{attribute 'enable_dynamic_creation'}
{attribute 'no_explicit_call' := 'direct call for this function block is not allowed'}
FUNCTION_BLOCK FB_ErrorTimestamp IMPLEMENTS I_ErrorTimestamp
VAR
	_nTimestamp : ULINT;
END_VAR

// Retrieves the timestamp as a combined date and time value.
METHOD AsDateTime : DT // The combined date and time value as a DT (Date and Time).
VAR_INPUT
END_VAR
AsDateTime := TO_DT(THIS^._nTimestamp/1000);
END_METHOD

// Retrieves the date part of the timestamp.
METHOD GetDate : DATE // The date part of the timestamp.
VAR_INPUT
END_VAR
GetDate := TO_DATE(THIS^._nTimestamp/1000);
END_METHOD

// Retrieves the time of day part of the timestamp.
METHOD GetTimeOfDay : TOD // The time of day part of the timestamp.
VAR_INPUT
END_VAR
GetTimeOfDay := TO_TOD(THIS^._nTimestamp MOD 86400000);
END_METHOD

// The raw timestamp value which represents the number of milliseconds since Thursday, 1.1.1970 00:00:00.000.
// [get] Returns the raw timestamp value.
// [set] Sets the raw timestamp value.
PROPERTY Raw : ULINT
GET
Raw := THIS^._nTimestamp;
END_GET
SET
THIS^._nTimestamp := Raw;
END_SET
END_PROPERTY

END_FUNCTION_BLOCK

(* stored: Version 1.1.0.1
   POU FB_ErrorTimestamp: Id {3006405e-b4c3-05aa-13ca-bc7db81a079f}, SpecialFunc None
   Method AsDateTime: Id {f8abec48-c1cf-0a93-07f7-ae776de09770}
   Method GetDate: Id {8828e0c1-8f04-0d4e-3a6f-d1c9f2a8f29b}
   Method GetTimeOfDay: Id {d08f581d-15b3-093b-15d0-177ad6073580}
   Property Raw: Id {da7c7bb0-400d-0d20-0daa-990da27b9d05}
   Get Get: Id {21722fe0-3607-0632-1491-3954b191ad41}
   Set Set: Id {0d1c1a45-8759-0f1c-3890-954be06c6a88} *)
